(* IEC 61131-3 sources: eCockpitGit/test_project/src/%F%00 Library/%F%Common Functions/%F%Networking/%ITF%ITF_TCPControllerManagement, 2 files *)

(* ---- %METH%onClose.st ---- *)
//Called when controller conection is closed
// |**Version**|**Author**| **Date** |**Changes**
// | 1         | NSN      | 20-05-22 | Creation
METHOD onClose
VAR_INPUT
	index			:WORD;				//Index set to controller
END_VAR
VAR_IN_OUT
	controller		:FB_TCPController;	//Controller which is closed
END_VAR
(*%!%__DELIMITER__%!%*)

(* ---- %METH%onOpen.st ---- *)
//Called when controller conection is opened
// |**Version**|**Author**| **Date** |**Changes**
// | 1         | NSN      | 20-05-22 | Creation
METHOD onOpen: BOOL
VAR_INPUT
	index			:WORD;				//Index set to controller
END_VAR
VAR_IN_OUT
	controller		:FB_TCPController;	//Controller which is closed
END_VAR
(*%!%__DELIMITER__%!%*)
